// TIA Portal V17 export
// export: Created 2023-02-25T16:31:53.1733938Z, ExportSetting WithDefaults, DisplayName Totally Integrated Automation Portal, DisplayVersion V17, DisplayName TIA Portal Openness, DisplayVersion V17, DisplayName TIA Portal Version Control Interface, DisplayVersion V17, DisplayName TIA Portal Test Suite Advanced, DisplayVersion V17, DisplayName STEP 7 Professional, DisplayVersion V17, DisplayName SIMATIC Energy Suite, DisplayVersion V17, DisplayName STEP 7 Safety, DisplayVersion V17, DisplayName WinCC Professional, DisplayVersion V17
FUNCTION "LOG_ButtonsManualLight" : Void   // FC9, LAD
{ S7_Optimized_Access := 'TRUE' }
VERSION : 0.1
// stored: AutoNumber true, IsIECCheckEnabled false, SetENOAutomatically false, UDAEnableTagReadback false
BEGIN

REGION Network 1: Button C1 light
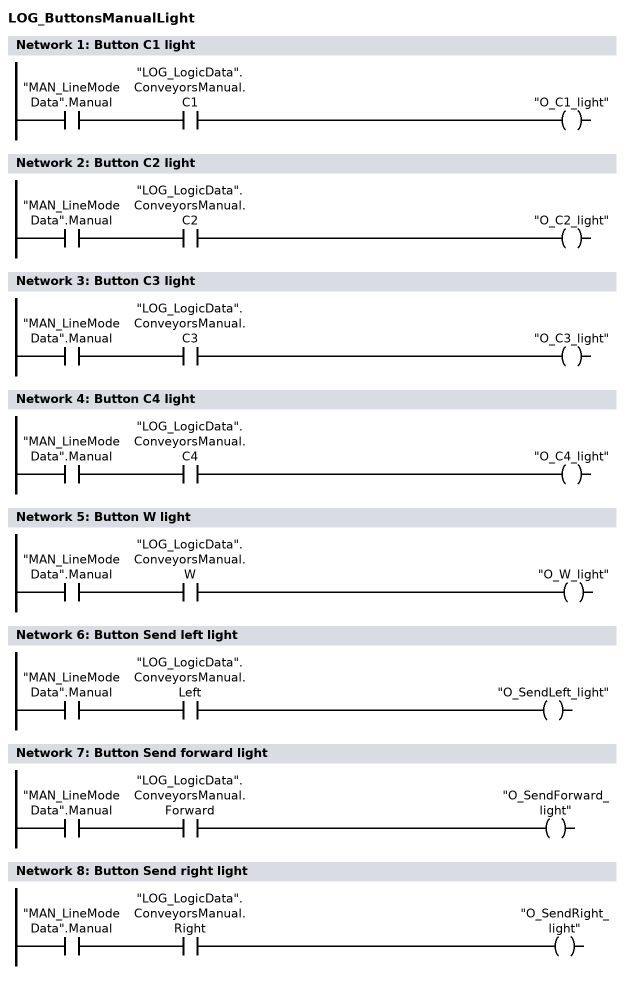
   RUNG wire#powerrail
      Contact( "MAN_LineModeData".Manual )
      Contact( "LOG_LogicData".ConveyorsManual.C1 )
      Coil( "O_C1_light" )
   END_RUNG
   // the same network as SCL:
   "O_C1_light" := "MAN_LineModeData".Manual AND "LOG_LogicData".ConveyorsManual.C1;
END_REGION

REGION Network 2: Button C2 light
   RUNG wire#powerrail
      Contact( "MAN_LineModeData".Manual )
      Contact( "LOG_LogicData".ConveyorsManual.C2 )
      Coil( "O_C2_light" )
   END_RUNG
   // the same network as SCL:
   "O_C2_light" := "MAN_LineModeData".Manual AND "LOG_LogicData".ConveyorsManual.C2;
END_REGION

REGION Network 3: Button C3 light
   RUNG wire#powerrail
      Contact( "MAN_LineModeData".Manual )
      Contact( "LOG_LogicData".ConveyorsManual.C3 )
      Coil( "O_C3_light" )
   END_RUNG
   // the same network as SCL:
   "O_C3_light" := "MAN_LineModeData".Manual AND "LOG_LogicData".ConveyorsManual.C3;
END_REGION

REGION Network 4: Button C4 light
   RUNG wire#powerrail
      Contact( "MAN_LineModeData".Manual )
      Contact( "LOG_LogicData".ConveyorsManual.C4 )
      Coil( "O_C4_light" )
   END_RUNG
   // the same network as SCL:
   "O_C4_light" := "MAN_LineModeData".Manual AND "LOG_LogicData".ConveyorsManual.C4;
END_REGION

REGION Network 5: Button W light
   RUNG wire#powerrail
      Contact( "MAN_LineModeData".Manual )
      Contact( "LOG_LogicData".ConveyorsManual.W )
      Coil( "O_W_light" )
   END_RUNG
   // the same network as SCL:
   "O_W_light" := "MAN_LineModeData".Manual AND "LOG_LogicData".ConveyorsManual.W;
END_REGION

REGION Network 6: Button Send left light
   RUNG wire#powerrail
      Contact( "MAN_LineModeData".Manual )
      Contact( "LOG_LogicData".ConveyorsManual.Left )
      Coil( "O_SendLeft_light" )
   END_RUNG
   // the same network as SCL:
   "O_SendLeft_light" := "MAN_LineModeData".Manual AND "LOG_LogicData".ConveyorsManual.Left;
END_REGION

REGION Network 7: Button Send forward light
   RUNG wire#powerrail
      Contact( "MAN_LineModeData".Manual )
      Contact( "LOG_LogicData".ConveyorsManual.Forward )
      Coil( "O_SendForward_light" )
   END_RUNG
   // the same network as SCL:
   "O_SendForward_light" := "MAN_LineModeData".Manual AND "LOG_LogicData".ConveyorsManual.Forward;
END_REGION

REGION Network 8: Button Send right light
   RUNG wire#powerrail
      Contact( "MAN_LineModeData".Manual )
      Contact( "LOG_LogicData".ConveyorsManual.Right )
      Coil( "O_SendRight_light" )
   END_RUNG
   // the same network as SCL:
   "O_SendRight_light" := "MAN_LineModeData".Manual AND "LOG_LogicData".ConveyorsManual.Right;
END_REGION
END_FUNCTION
